PROGRAM AXES_CYCLE
VAR
END_VAR

GRP1();

ACTION GRP1:
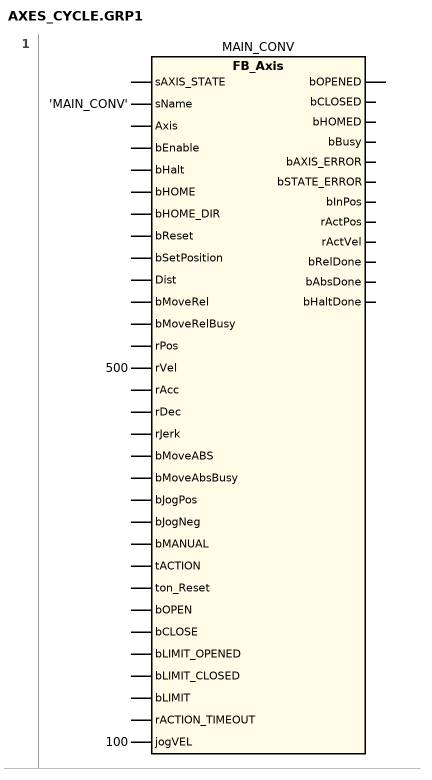
// NETWORK 1
MAIN_CONV(sName := 'MAIN_CONV', rVel := 500, jogVEL := 100); // FB_Axis

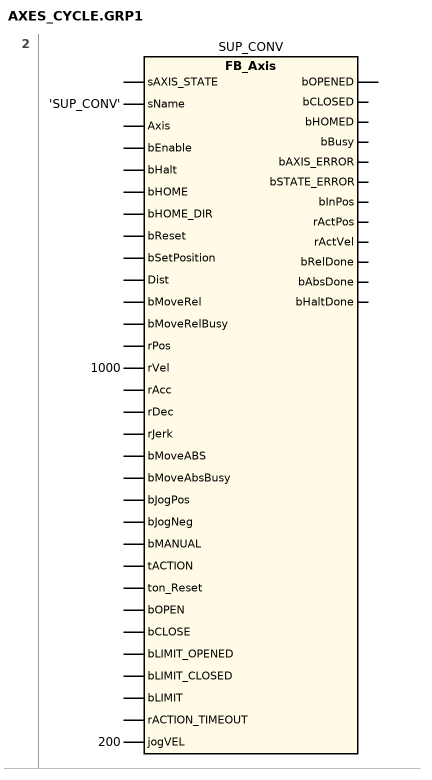
// NETWORK 2
SUP_CONV(sName := 'SUP_CONV', rVel := 1000, jogVEL := 200); // FB_Axis

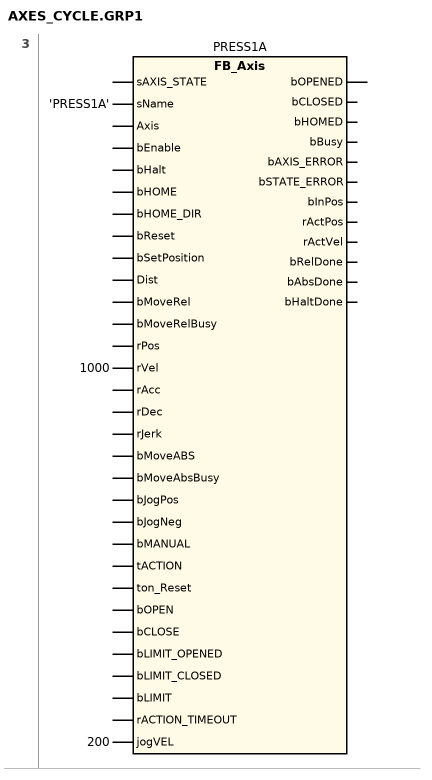
// NETWORK 3
PRESS1A(sName := 'PRESS1A', rVel := 1000, jogVEL := 200); // FB_Axis

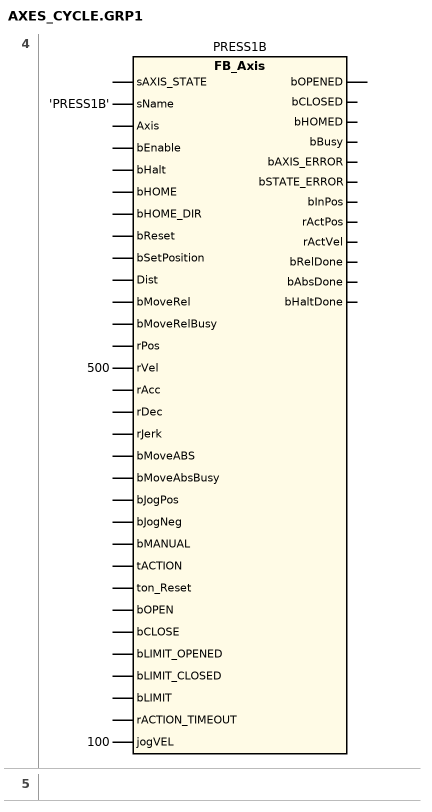
// NETWORK 4
PRESS1B(sName := 'PRESS1B', rVel := 500, jogVEL := 100); // FB_Axis

// NETWORK 5
END_ACTION

END_PROGRAM

(* stored: Version 1.1.0.1, ProductVersion 3.1.4024.12
   POU AXES_CYCLE: Id {9cd0cba8-0116-4d06-bcad-bfddb259f9ba}, SpecialFunc None
   Action GRP1: Id {c92a8f88-fc9a-4b1d-835c-ccf46ea4c98c} *)
